FUNCTION_BLOCK FB_MirrorCoatingProtectionScaledPositions
VAR_INPUT
	bMirrorIn :BOOL; //Mirror is in the In position
	rCurrentEncoderPosition : REAL; // Current encoder position
	neVRange : WORD; // Current ev range from stCurrentBeamParams	
	sDevName : STRING := ''; // Device name	
	rFirstCoatingPosition : REAL; // Encoder count/position for the coating 
	rFirstCoatingPositionTolerance : REAL; // position +/- tolerance 
	nFirstCoatingBitmask : WORD; // Bitmask for upper coating
	sFirstCoatingType : STRING := ''; // Type of coating
	rSecondCoatingPosition : REAL; // Encoder count/position for the coating 
	rSecondCoatingPositionTolerance : REAL; // position +/- tolerance 
	nSecondCoatingBitmask : WORD; // Bitmask for upper coating
	sSecondCoatingType : STRING := ''; // Type of coating
	bAutoClear : BOOL;
END_VAR
VAR_OUTPUT
END_VAR
VAR_IN_OUT
	FFO : FB_HardwareFFOutput;
END_VAR
VAR
	ffFirstCoating: FB_FastFault;
	ffSecondCoating: FB_FastFault;	
	bInit : BOOL :=TRUE;
END_VAR

IF  bInit THEN
	ffFirstCoating.i_Desc := CONCAT(sFirstCoatingType, ' mirror coating incompatible with beam photon energy');
	ffFirstCoating.i_DevName := sDevName;
	
	ffSecondCoating.i_Desc := CONCAT(sSecondCoatingType, ' mirror coating incompatible with beam photon energy');
	ffSecondCoating.i_DevName := sDevName;
	bInit := FALSE;
END_IF
IF (bMirrorIn) THEN
	IF (rCurrentEncoderPosition >= rFirstCoatingPosition - rFirstCoatingPositionTolerance) AND (rCurrentEncoderPosition <= rFirstCoatingPosition + rFirstCoatingPositionTolerance)  THEN
		ffFirstCoating.i_xOK := (neVRange AND nFirstCoatingBitmask) = neVRange; 
		ffSecondCoating.i_xOK := TRUE;
	ELSIF (rCurrentEncoderPosition >= rSecondCoatingPosition - rSecondCoatingPositionTolerance) AND (rCurrentEncoderPosition <= rSecondCoatingPosition + rSecondCoatingPositionTolerance)  THEN
		ffSecondCoating.i_xOK := (neVRange AND nSecondCoatingBitmask) = neVRange; 
		ffFirstCoating.i_xOK := TRUE;
	ELSE
		ffFirstCoating.i_xOK := FALSE;
		ffSecondCoating.i_xOK := FALSE;
	END_IF
ELSE 
	ffFirstCoating.i_xOK := TRUE;
	ffSecondCoating.i_xOK := TRUE;
END_IF
ffFirstCoating(
		i_xAutoReset := bAutoClear,
		i_TypeCode := 16#601,
	    io_fbFFHWO:=FFO);
		
ffSecondCoating(
		i_xAutoReset := bAutoClear,
		i_TypeCode := 16#601,
	    io_fbFFHWO:=FFO);

END_FUNCTION_BLOCK

(* stored: Version 1.1.0.1, ProductVersion 3.1.4024.6
   POU FB_MirrorCoatingProtectionScaledPositions: Id {d10577b5-3cca-4b2d-9575-3f7b707b5b15}, SpecialFunc None *)
